// TIA Portal V17 export
// export: Created 2025-03-07T09:19:23.0922074Z, ExportSetting WithDefaults, DisplayName Totally Integrated Automation Portal, DisplayVersion V17 Update 8, DisplayName TIA Portal Openness, DisplayVersion V17 Update 8, DisplayName TIA Portal Version Control Interface, DisplayVersion V17, DisplayName SINAMICS Startdrive Advanced, DisplayVersion V17 SP2, DisplayName SINAMICS Startdrive G110M, G120, G120C, G120D, G120P, G115D, DisplayVersion V17 SP2, DisplayName SINAMICS Startdrive G130, G150, S120, S150, SINAMICS MV, S210, DisplayVersion V17 SP2, DisplayName STEP 7 Professional, DisplayVersion V17 Update 8, DisplayName SINUMERIK ONE STEP 7 Toolbox, DisplayVersion V17 Update 12, DisplayName SINUMERIK 840D sl STEP 7 Toolbox, DisplayVersion V17 Update 12, DisplayName STEP 7 Safety, DisplayVersion V17 Update 6, DisplayName WinCC Advanced, DisplayVersion V17 Update 8
VAR_GLOBAL   // PLC tag table "TAGS_IO_CYLINDERS_CLADDING"
   "/////_SAFETY_BRAKES_/////" AT %M1200.0 : Bool;   // /////_SAFETY_BRAKES_/////
   SAFETY_BRAKE_AXIS_Z13_BLCKD_I AT %I570.5 : Bool;   // AXIS Z13 BRAKE BLOCKED INPUT
   SAFETY_BRAKE_AXIS_Z13_UNBLCKD_I AT %I570.6 : Bool;   // AXIS Z13 BRAKE UNBLOCKED INPUT
   SAFETY_BRAKE_AXIS_Z13_MAINT_BLCKD_I AT %M1200.3 : Bool;   // SAFETY BRAKE AXIS Z13 MAINTENANCE BRAKE BLOCKED INPUT
   SAFETY_BRAKE_AXIS_Z13_MAINT_UNBLCKD_I AT %M1200.4 : Bool;   // SAFETY BRAKE AXIS Z13 MAINTENANCE BRAKE UNBLOCKED INPUT
   SAFETY_BRAKE_AXIS_Z13_BLCK_Q AT %M1200.5 : Bool;   // SAFETY BRAKE AXIS Z13 BLOCK OUTPUT
   SAFETY_BRAKE_AXIS_Z23_BLCKD_I AT %I1570.5 : Bool;   // SAFETY BRAKE AXIS Z23 BLOCKED INPUT
   SAFETY_BRAKE_AXIS_Z23_UNBLCKD_I AT %I1570.6 : Bool;   // SAFETY BRAKE AXIS Z23 UNBLOCKED INPUT
   SAFETY_BRAKE_AXIS_Z23_MAINT_BLCKD_I AT %M1201.1 : Bool;   // SAFETY BRAKE AXIS Z23 MAINTENANCE BRAKE BLOCKED INPUT
   SAFETY_BRAKE_AXIS_Z23_MAINT_UNBLCKD_I AT %M1201.2 : Bool;   // SAFETY BRAKE AXIS Z23 MAINTENANCE BRAKE UNBLOCKED INPUT
   SAFETY_BRAKE_AXIS_Z23_BLCK_Q AT %M1201.3 : Bool;   // SAFETY BRAKE AXIS Z23 BLOCK OUTPUT
   "/////_UP_SEALING_U01_STRUCTURE_/////" AT %M1201.5 : Bool;   // /////_UP_SEALING_U01_STRUCTURE_/////
   UP_SEALING_U01_OPND_I_1 AT %I490.2 : Bool;   // UP SEALING UNIT 01 STRUCTURE OPENED INPUT 1
   UP_SEALING_U01_OPND_I_2 AT %I490.4 : Bool;   // UP SEALING UNIT 01 STRUCTURE OPENED INPUT 2
   UP_SEALING_U01_OPND_I_3 AT %I470.4 : Bool;   // UP SEALING UNIT 01 STRUCTURE OPENED INPUT 3
   UP_SEALING_U01_OPND_I_4 AT %I470.6 : Bool;   // UP SEALING UNIT 01 STRUCTURE OPENED INPUT 4
   UP_SEALING_U01_CLSD_I_1 AT %I490.3 : Bool;   // UP SEALING UNIT 01 STRUCTURE CLOSED INPUT 1
   UP_SEALING_U01_CLSD_I_2 AT %I490.5 : Bool;   // UP SEALING UNIT 01 STRUCTURE CLOSED INPUT 2
   UP_SEALING_U01_CLSD_I_3 AT %I470.5 : Bool;   // UP SEALING UNIT 01 STRUCTURE CLOSED INPUT 3
   UP_SEALING_U01_CLSD_I_4 AT %I470.7 : Bool;   // UP SEALING UNIT 01 STRUCTURE CLOSED INPUT 4
   "/////_DOWN_SEALING_U01_STRUCTURE_/////" AT %M1203.0 : Bool;   // /////_DOWN_SEALING_U01_STRUCTURE_/////
   DOWN_SEALING_U01_OPND_I_1 AT %M1203.1 : Bool;   // DOWN SEALING UNIT 01 STRUCTURE OPENED INPUT 1
   DOWN_SEALING_U01_OPND_I_2 AT %M1203.2 : Bool;   // DOWN SEALING UNIT 01 STRUCTURE OPENED INPUT 2
   DOWN_SEALING_U01_OPND_I_3 AT %I490.7 : Bool;   // DOWN SEALING UNIT 01 STRUCTURE OPENED INPUT 3
   DOWN_SEALING_U01_OPND_I_4 AT %I480.1 : Bool;   // DOWN SEALING UNIT 01 STRUCTURE OPENED INPUT 4
   DOWN_SEALING_U01_CLSD_I_1 AT %M1203.5 : Bool;   // DOWN SEALING UNIT 01 STRUCTURE CLOSED INPUT 1
   DOWN_SEALING_U01_CLSD_I_2 AT %M1203.6 : Bool;   // DOWN SEALING UNIT 01 STRUCTURE CLOSED INPUT 2
   DOWN_SEALING_U01_CLSD_I_3 AT %I490.6 : Bool;   // DOWN SEALING UNIT 01 STRUCTURE CLOSED INPUT 3
   DOWN_SEALING_U01_CLSD_I_4 AT %I480.0 : Bool;   // DOWN SEALING UNIT 01 STRUCTURE CLOSED INPUT 4
   DOWN_SEALING_U01_OPEN_Q AT %Q72.3 : Bool;   // DOWN SEALING UNIT 01 STRUCTURE OPEN OUTPUT
   DOWN_SEALING_U01_CLOSE_Q AT %Q72.2 : Bool;   // DOWN SEALING UNIT 01 STRUCTURE CLOSE OUTPUT
   "/////_UNIT_01_BEAM_SAMPLER/////" AT %M1207.1 : Bool;   // /////_UNIT_01_BEAM_SAMPLER/////
   U01_ST4_BEAM_SAMPLER_BLOW_I AT %M1207.2 : Bool;   // UNIT 01 BEAM SAMPLER BLOWING INPUT
   U01_ST4_BEAM_SAMPLER_PRESSURIZED_I AT %M1207.3 : Bool;   // UNIT 01 BEAM SAMPLER PRESSURIZED INPUT
   U01_ST4_BEAM_SAMPLER_BLOW_Q AT %M1207.4 : Bool;   // UNIT 01 BEAM SAMPLER BLOW OUTPUT STATION 4
   "/////_UNIT_01_DUST_EXTRACTION_1/////" AT %M1207.5 : Bool;   // /////_UNIT_01_DUST_EXTRACTION_1/////
   U01_DUST_EXTRAC_1_SWTCHD_ON_I AT %M1207.6 : Bool;   // UNIT 01 DUST EXTRACCION 1 SWITCHED ON INPUT (Flow Present)
   U01_DUST_EXTRAC_1_SWTCHD_OFF_I AT %M1207.7 : Bool;   // UNIT 01 DUST EXTRACCION 1 SWITCHED OFF INPUT
   U01_DUST_EXTRAC_1_SWTCH_OFF_Q AT %M1208.1 : Bool;   // UNIT 01 DUST EXTRACCION 1 SWITCH OFF OUTPUT
   "/////_UNIT_01_DUST_EXTRACTION_2/////" AT %M1208.2 : Bool;   // /////_UNIT_01_DUST_EXTRACTION_2/////
   U01_DUST_EXTRAC_2_SWTCHD_ON_I AT %M1208.3 : Bool;   // UNIT 01 DUST EXTRACCION 2 SWITCHED ON INPUT (Flow Present)
   U01_DUST_EXTRAC_2_SWTCHD_OFF_I AT %M1208.4 : Bool;   // UNIT 01 DUST EXTRACCION 2 SWITCHED OFF INPUT
   U01_DUST_EXTRAC_2_SWTCH_ON_Q AT %M1208.5 : Bool;   // UNIT 01 DUST EXTRACCION 2 SWITCH ON OUTPUT
   U01_DUST_EXTRAC_2_SWTCH_OFF_Q AT %M1208.6 : Bool;   // UNIT 01 DUST EXTRACCION 2 SWITCH OFF OUTPUT
   "/////_UNIT_01_DUST_EXTRACTION_3/////" AT %M1208.7 : Bool;   // /////_UNIT_01_DUST_EXTRACTION_3/////
   U01_DUST_EXTRAC_3_SWTCHD_ON_I AT %M1209.0 : Bool;   // UNIT 01 DUST EXTRACCION 3 SWITCHED ON INPUT (Flow Present)
   U01_DUST_EXTRAC_3_SWTCHD_OFF_I AT %M1209.1 : Bool;   // UNIT 01 DUST EXTRACCION 3 SWITCHED OFF INPUT
   U01_DUST_EXTRAC_3_SWTCH_OFF_Q AT %M1209.3 : Bool;   // UNIT 01 DUST EXTRACCION 3 SWITCH OFF OUTPUT
   "/////_UNIT_01_DUST_EXTRACTION_4/////" AT %M1209.4 : Bool;   // /////_UNIT_01_DUST_EXTRACTION_4/////
   U01_DUST_EXTRAC_4_SWTCHD_ON_I AT %M1209.5 : Bool;   // UNIT 01 DUST EXTRACCION 4 SWITCHED ON INPUT (Flow Present)
   U01_DUST_EXTRAC_4_SWTCHD_OFF_I AT %M1209.6 : Bool;   // UNIT 01 DUST EXTRACCION 4 SWITCHED OFF INPUT
   U01_DUST_EXTRAC_4_SWTCH_OFF_Q AT %M1210.0 : Bool;   // UNIT 01 DUST EXTRACCION 4 SWITCH OFF OUTPUT
   "/////_UNIT_01_ANGULAR_LOCATOR_/////" AT %M1210.6 : Bool;
   U01_ANGULAR_LOCATOR_LCTD_I AT %I578.0 : Bool;
   U01_ANGULAR_LOCATOR_RTND_I AT %I578.1 : Bool;
   U01_ANGULAR_LOCATOR_LCT_Q AT %Q74.0 : Bool;   // UNIT 01 ANGULAR LOCATOR LOCATE OUTPUT
   U01_ANGULAR_LOCATOR_RTN_Q AT %Q74.1 : Bool;   // UNIT 01 ANGULAR LOCATOR RETURN OUTPUT
   "/////_UNIT_01_AXIAL_LOCATOR_/////" AT %M1211.3 : Bool;
   U01_AXIAL_LOCATOR_LCTD_I AT %I578.2 : Bool;
   U01_AXIAL_LOCATOR_RTND_I AT %I578.3 : Bool;
   U01_AXIAL_LOCATOR_LCT_Q AT %Q74.2 : Bool;   // UNIT 01 AXIAL LOCATOR LOCATE OUTPUT
   U01_AXIAL_LOCATOR_RTN_Q AT %Q74.3 : Bool;   // UNIT 01 AXIAL LOCATOR RETURN OUTPUT
   "/////_UNIT_01_STATION_4_BRUSH/////" AT %M1212.0 : Bool;   // /////_UNIT_01_STATION_4_BRUSH/////
   U01_ST4_BRUSH_LCTD_I AT %M1212.1 : Bool;   // UNIT 01 STATION 4 BRUSH LOCATED INPUT
   U01_ST4_BRUSH_RTND_I AT %M1212.2 : Bool;   // UNIT 01 STATION 4 BRUSH RETURNED INPUT
   U01_ST4_BRUSH_LCT_Q AT %M1212.3 : Bool;
   U01_ST4_BRUSH_RTN_Q AT %M1212.4 : Bool;
   "/////_UP_SEALING_U02_STRUCTURE_/////" AT %M1212.5 : Bool;   // /////_UP_SEALING_U02_STRUCTURE_/////
   UP_SEALING_U02_OPND_I_1 AT %I1490.2 : Bool;   // UP SEALING UNIT 02 STRUCTURE OPENED INPUT 1
   UP_SEALING_U02_OPND_I_2 AT %I1490.4 : Bool;   // UP SEALING UNIT 02 STRUCTURE OPENED INPUT 2
   UP_SEALING_U02_OPND_I_3 AT %I1470.4 : Bool;   // UP SEALING UNIT 02 STRUCTURE OPENED INPUT 3
   UP_SEALING_U02_OPND_I_4 AT %I1470.6 : Bool;   // UP SEALING UNIT 02 STRUCTURE OPENED INPUT 4
   UP_SEALING_U02_CLSD_I_1 AT %I1490.3 : Bool;   // UP SEALING UNIT 02 STRUCTURE CLOSED INPUT 1
   UP_SEALING_U02_CLSD_I_2 AT %I1490.5 : Bool;   // UP SEALING UNIT 02 STRUCTURE CLOSED INPUT 2
   UP_SEALING_U02_CLSD_I_3 AT %I1470.5 : Bool;   // UP SEALING UNIT 02 STRUCTURE CLOSED INPUT 3
   UP_SEALING_U02_CLSD_I_4 AT %I1470.7 : Bool;   // UP SEALING UNIT 02 STRUCTURE CLOSED INPUT 4
   "/////_DOWN_SEALING_U02_STRUCTURE_/////" AT %M1214.0 : Bool;   // /////_DOWN_SEALING_U02_STRUCTURE_/////
   DOWN_SEALING_U02_OPND_I_1 AT %M1214.1 : Bool;   // DOWN SEALING UNIT 02 STRUCTURE OPENED INPUT 1
   DOWN_SEALING_U02_OPND_I_2 AT %M1214.2 : Bool;   // DOWN SEALING UNIT 02 STRUCTURE OPENED INPUT 2
   DOWN_SEALING_U02_OPND_I_3 AT %I1490.7 : Bool;   // DOWN SEALING UNIT 02 STRUCTURE OPENED INPUT 3
   DOWN_SEALING_U02_OPND_I_4 AT %I1480.1 : Bool;   // DOWN SEALING UNIT 02 STRUCTURE OPENED INPUT 4
   DOWN_SEALING_U02_CLSD_I_1 AT %M1214.5 : Bool;   // DOWN SEALING UNIT 02 STRUCTURE CLOSED INPUT 1
   DOWN_SEALING_U02_CLSD_I_2 AT %M1214.6 : Bool;   // DOWN SEALING UNIT 02 STRUCTURE CLOSED INPUT 2
   DOWN_SEALING_U02_CLSD_I_3 AT %I1490.6 : Bool;   // DOWN SEALING UNIT 02 STRUCTURE CLOSED INPUT 3
   DOWN_SEALING_U02_CLSD_I_4 AT %I1480.0 : Bool;   // DOWN SEALING UNIT 02 STRUCTURE CLOSED INPUT 4
   DOWN_SEALING_U02_OPEN_Q AT %Q1072.3 : Bool;   // DOWN SEALING UNIT 02 STRUCTURE OPEN OUTPUT
   DOWN_SEALING_U02_CLOSE_Q AT %Q1072.2 : Bool;   // DOWN SEALING UNIT 02 STRUCTURE CLOSE OUTPUT
   "/////_UNIT_02_BEAM_SAMPLER/////" AT %M1215.3 : Bool;   // /////_UNIT_02_BEAM_SAMPLER/////
   U02_ST4_BEAM_SAMPLER_BLOW_I AT %M1215.4 : Bool;   // UNIT 02 BEAM SAMPLER BLOWING INPUT
   U02_ST4_BEAM_SAMPLER_PRESSURIZED_I AT %M1215.5 : Bool;   // UNIT 02 BEAM SAMPLER PRESSURIZED INPUT
   U02_ST4_BEAM_SAMPLER_BLOW_Q AT %M1215.6 : Bool;   // UNIT 01 BEAM SAMPLER BLOW OUTPUT STATION 4
   "/////_UNIT_02_DUST_EXTRACTION_1_/////" AT %M1215.7 : Bool;   // /////_UNIT_02_DUST_EXTRACTION_1/////
   U02_DUST_EXTRAC_1_SWTCHD_ON_I AT %M1216.0 : Bool;   // UNIT 02 DUST EXTRACCION 1 SWITCHED ON INPUT (Flow Present)
   U02_DUST_EXTRAC_1_SWTCHD_OFF_I AT %M1216.1 : Bool;   // UNIT 02 DUST EXTRACCION 1 SWITCHED OFF INPUT
   U02_DUST_EXTRAC_1_SWTCH_OFF_Q AT %M1216.3 : Bool;   // UNIT 02 DUST EXTRACCION 1 SWITCH OFF OUTPUT
   "/////_UNIT_02_DUST_EXTRACTION_2_/////" AT %M1216.4 : Bool;   // /////_UNIT_02_DUST_EXTRACTION_2/////
   U02_DUST_EXTRAC_2_SWTCHD_ON_I AT %M1216.5 : Bool;   // UNIT 02 DUST EXTRACCION 2 SWITCHED ON INPUT (Flow Present)
   U02_DUST_EXTRAC_2_SWTCHD_OFF_I AT %M1216.6 : Bool;   // UNIT 02 DUST EXTRACCION 2 SWITCHED OFF INPUT
   U02_DUST_EXTRAC_2_SWTCH_ON_Q AT %M1216.7 : Bool;   // UNIT 02 DUST EXTRACCION 2 SWITCH ON OUTPUT
   U02_DUST_EXTRAC_2_SWTCH_OFF_Q AT %M1217.0 : Bool;   // UNIT 02 DUST EXTRACCION 2 SWITCH OFF OUTPUT
   "/////_UNIT_02_DUST_EXTRACTION_3_/////" AT %M1217.1 : Bool;   // /////_UNIT_02_DUST_EXTRACTION_3/////
   U02_DUST_EXTRAC_3_SWTCHD_ON_I AT %M1217.2 : Bool;   // UNIT 02 DUST EXTRACCION 3 SWITCHED ON INPUT (Flow Present)
   U02_DUST_EXTRAC_3_SWTCHD_OFF_I AT %M1217.3 : Bool;   // UNIT 02 DUST EXTRACCION 3 SWITCHED OFF INPUT
   U02_DUST_EXTRAC_3_SWTCH_ON_Q AT %Q1073.2 : Bool;   // UNIT 02 DUST EXTRACCION 3 SWITCH ON OUTPUT
   U02_DUST_EXTRAC_3_SWTCH_OFF_Q AT %M1217.5 : Bool;   // UNIT 02 DUST EXTRACCION 3 SWITCH OFF OUTPUT
   "/////_UNIT_02_DUST_EXTRACTION_4_/////" AT %M1217.6 : Bool;   // /////_UNIT_02_DUST_EXTRACTION_4/////
   U02_DUST_EXTRAC_4_SWTCHD_ON_I AT %M1217.7 : Bool;   // UNIT 02 DUST EXTRACCION 4 SWITCHED ON INPUT (Flow Present)
   U02_DUST_EXTRAC_4_SWTCHD_OFF_I AT %M1218.0 : Bool;   // UNIT 02 DUST EXTRACCION 4 SWITCHED OFF INPUT
   U02_DUST_EXTRAC_4_SWTCH_OFF_Q AT %M1218.2 : Bool;   // UNIT 02 DUST EXTRACCION 4 SWITCH OFF OUTPUT
   "/////_UNIT_02_ANGULAR_LOCATOR_/////" AT %M1219.5 : Bool;
   U02_ANGULAR_LOCATOR_LCTD_I AT %I1578.0 : Bool;
   U02_ANGULAR_LOCATOR_RTND_I AT %I1578.1 : Bool;
   U02_ANGULAR_LOCATOR_LCT_Q AT %Q1074.0 : Bool;   // UNIT 01 ANGULAR LOCATOR LOCATE OUTPUT
   U02_ANGULAR_LOCATOR_RTN_Q AT %Q1074.1 : Bool;   // UNIT 01 ANGULAR LOCATOR RETURN OUTPUT
   "/////_UNIT_02_AXIAL_LOCATOR_/////" AT %M1220.2 : Bool;
   U02_AXIAL_LOCATOR_LCTD_I AT %I1578.2 : Bool;
   U02_AXIAL_LOCATOR_RTND_I AT %I1578.3 : Bool;
   U02_AXIAL_LOCATOR_LCT_Q AT %Q1074.2 : Bool;   // UNIT 01 AXIAL LOCATOR LOCATE OUTPUT
   U02_AXIAL_LOCATOR_RTN_Q AT %Q1074.3 : Bool;   // UNIT 01 AXIAL LOCATOR RETURN OUTPUT
   "/////_UNIT_02_STATION_4_BRUSH/////" AT %M1220.7 : Bool;   // /////_UNIT_02_STATION_4_BRUSH/////
   U02_ST4_BRUSH_LCTD_I AT %M1221.0 : Bool;   // UNIT 02 STATION 4 BRUSH LOCATED INPUT
   U02_ST4_BRUSH_RTND_I AT %M1221.1 : Bool;   // UNIT 02 STATION 4 BRUSH RETURNED INPUT
   U02_ST4_BRUSH_LCT_Q AT %Q1075.6 : Bool;   // UNIT 02 STATION 4 BRUSH LOCATE OUTPUT
   U02_ST4_BRUSH_RTN_Q AT %Q1075.7 : Bool;   // UNIT 02 STATION 4 BRUSH RETURN OUTPUT
   U01_HAT_UP_DOWN AT %I480.7 : Bool;   // UNIT 01 STATION 1 HAT UP / HAT DOWN
   U02_HAT_UP_DOWN AT %I1480.7 : Bool;   // UNIT 02 HAT UP / HAT DOWN
   U02_STA_1_PART_PRESENT AT %I1480.6 : Bool;   // UNIT 02 STATION 1 PART PRESENT
   UP_SEALING_U02_OPEN_Q AT %Q1072.4 : Bool;   // UP SEALING UNIT 02 STRUCTURE CLOSE OUTPUT
   UP_SEALING_U02_CLOSE_Q AT %Q1072.5 : Bool;   // UP SEALING UNIT 02 STRUCTURE OPEN OUTPUT
   U01_DUST_EXTRAC_4_SWTCH_ON_Q AT %Q66.0 : Bool;   // UNIT 01 DUST EXTRACCION 4 SWITCH ON OUTPUT
   UP_SEALING_U01_CLOSE_Q AT %Q72.5 : Bool;   // UP SEALING UNIT 01 STRUCTURE CLOSE (MOVE DOWN) OUTPUT
   UP_SEALING_U01_OPEN_Q AT %Q72.4 : Bool;   // UP SEALING UNIT 01 STRUCTURE OPEN (MOVE UP) OUTPUT
   U01_DUST_EXTRAC_1_SWTCH_ON_Q AT %Q66.2 : Bool;   // UNIT 01 DUST EXTRACCION 1 SWITCH ON OUTPUT
   SAFETY_BRAKE_AXIS_Z23_UNBLCK_Q AT %Q1072.6 : Bool;   // SAFETY BRAKE AXIS Z23 UNBLOCK OUTPUT
   SAFETY_BRAKE_AXIS_Z13_UNBLCK_Q AT %Q72.6 : Bool;   // SAFETY BRAKE AXIS Z13 UNBLOCK OUTPUT
   KF76_SAFE_VALVE_ON AT %Q72.0 : Bool;   // KF76 SAFETY VALVE ON
   U01_DUST_EXTRAC_3_SWTCH_ON_Q AT %Q66.6 : Bool;   // UNIT 01 DUST EXTRACCION 3 SWITCH ON OUTPUT
   U02_DUST_EXTRAC_1_SWTCH_ON_Q AT %Q1066.2 : Bool;   // UNIT 02 DUST EXTRACCION 1 SWITCH ON OUTPUT
   U01_STA_1_PART_PRESENT_NC AT %I481.6 : Bool;   // UNIT 01 STATION 1 PART PRESENT NC
   U01_STA_1_PART_PRESENT_NO AT %I480.6 : Bool;   // UNIT 01 STATION 1 PART PRESENT NO
   U02_DUST_EXTRAC_4_SWTCH_ON_Q AT %Q1066.0 : Bool;   // UNIT 02 DUST EXTRACCION 4 SWITCH ON OUTPUT
END_VAR
